FUNCTION_BLOCK SawmillSwitch (* goFB_ignore *)
  (* Standard: 61499-2 *)
  (* Version 0.1, 2017-00-16, hpea485, UOA *)
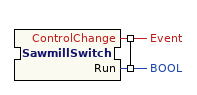
  EVENT_OUTPUT
    ControlChange WITH Run;
  END_EVENT
  VAR_OUTPUT
    Run : BOOL;
  END_VAR
  EC_STATES
    Start;
  END_STATES
END_FUNCTION_BLOCK
